INTERFACE IFuseChannelExtended EXTENDS __SYSTEM.IQueryInterface

PROPERTY DisabledByDI : BOOL
GET
END_GET
END_PROPERTY

PROPERTY DisabledByOutput : BOOL
GET
END_GET
END_PROPERTY

PROPERTY DisabledBySwitch : BOOL
GET
END_GET
END_PROPERTY

PROPERTY Overload : BOOL
GET
END_GET
END_PROPERTY

PROPERTY Overvoltage : BOOL
GET
END_GET
END_PROPERTY

PROPERTY ShortCircuit : BOOL
GET
END_GET
END_PROPERTY

PROPERTY StateDeviceSwitch : BOOL
GET
END_GET
END_PROPERTY

PROPERTY StateDigitalInput : BOOL
GET
END_GET
END_PROPERTY

PROPERTY Undervoltage : BOOL
GET
END_GET
END_PROPERTY

END_INTERFACE

(* stored: Version 1.1.0.1, ProductVersion 3.1.4024.6
   Itf IFuseChannelExtended: Id {7b497cb5-6c2a-4cb3-a667-b782d5b1f17b}
   Property DisabledByDI: Id {2e43ff6c-dd3e-44e3-a427-f36edfceb496}
   Get Get: Id {9b705708-dc8d-41a3-83b3-baf0c5839a8a}
   Property DisabledByOutput: Id {06b8701f-906a-472d-bbae-c2ecde8ab279}
   Get Get: Id {f6954428-c199-4f6a-9ed7-59f12d42fcc6}
   Property DisabledBySwitch: Id {09f48e97-25d0-4ee4-8e46-712cb2c7d9c1}
   Get Get: Id {8f1de88f-2062-4568-8b7d-d244392cb283}
   Property Overload: Id {fbe7e518-5c5f-47c5-992a-c862e483ecb0}
   Get Get: Id {c4b4135d-065f-476d-a1c5-98d3bf95523a}
   Property Overvoltage: Id {4af56bc4-7609-4ef9-99d7-1686048c1622}
   Get Get: Id {84507bc7-0b14-4d2e-a071-51ae3010cf85}
   Property ShortCircuit: Id {f68a74aa-e2fe-40d1-a5e6-9b32dfadd7c0}
   Get Get: Id {4bbb5072-dcf1-4f37-9f85-3c566e9dac22}
   Property StateDeviceSwitch: Id {f988186b-99af-43fc-b808-8ea699b58dbe}
   Get Get: Id {ab85e28e-2e82-43ed-a5d0-8dc267972367}
   Property StateDigitalInput: Id {a1fe8b4a-d0c5-4c31-a664-4a2de53f665f}
   Get Get: Id {365646ad-42a3-4531-9f12-e677d6e933ee}
   Property Undervoltage: Id {ca3da1b6-0f91-4a64-9901-114f83399d0d}
   Get Get: Id {145165e1-802d-42e2-b70f-cc8dd1b461b8} *)
